FUNCTION_BLOCK Gerador (* CAT Gerador AGC150 - 15 blocos - 74 vars *)
  (* Standard: 61499-2 *)
  (* Version 7.0, 13/05/2026, Claude, 74 tags essenciais AGC150 *)
  PACKAGE Hidryco.HidrycoLib;
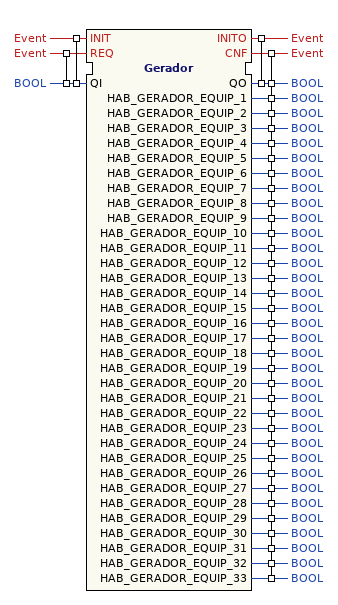
  EVENT_INPUT
    INIT WITH QI;
    REQ WITH QI;
  END_EVENT
  EVENT_OUTPUT
    INITO WITH QO;
    CNF WITH QO, HAB_GERADOR_EQUIP_4, HAB_GERADOR_EQUIP_5, HAB_GERADOR_EQUIP_6, HAB_GERADOR_EQUIP_7, HAB_GERADOR_EQUIP_8, HAB_GERADOR_EQUIP_9, HAB_GERADOR_EQUIP_10, HAB_GERADOR_EQUIP_11, HAB_GERADOR_EQUIP_12, HAB_GERADOR_EQUIP_13, HAB_GERADOR_EQUIP_14, HAB_GERADOR_EQUIP_15, HAB_GERADOR_EQUIP_16, HAB_GERADOR_EQUIP_17, HAB_GERADOR_EQUIP_18, HAB_GERADOR_EQUIP_19, HAB_GERADOR_EQUIP_20, HAB_GERADOR_EQUIP_21, HAB_GERADOR_EQUIP_22, HAB_GERADOR_EQUIP_23, HAB_GERADOR_EQUIP_24, HAB_GERADOR_EQUIP_25, HAB_GERADOR_EQUIP_26, HAB_GERADOR_EQUIP_27, HAB_GERADOR_EQUIP_28, HAB_GERADOR_EQUIP_29, HAB_GERADOR_EQUIP_30, HAB_GERADOR_EQUIP_31, HAB_GERADOR_EQUIP_32, HAB_GERADOR_EQUIP_33, HAB_GERADOR_EQUIP_1, HAB_GERADOR_EQUIP_2, HAB_GERADOR_EQUIP_3;
  END_EVENT
  VAR_INPUT
    QI : BOOL;
  END_VAR
  VAR_OUTPUT
    QO : BOOL;
    HAB_GERADOR_EQUIP_1 : BOOL; (* Habilitar equipamento 1 no gerador *)
    HAB_GERADOR_EQUIP_2 : BOOL; (* Habilitar equipamento 2 no gerador *)
    HAB_GERADOR_EQUIP_3 : BOOL; (* Habilitar equipamento 3 no gerador *)
    HAB_GERADOR_EQUIP_4 : BOOL; (* Habilitar equipamento 4 no gerador *)
    HAB_GERADOR_EQUIP_5 : BOOL; (* Habilitar equipamento 5 no gerador *)
    HAB_GERADOR_EQUIP_6 : BOOL; (* Habilitar equipamento 6 no gerador *)
    HAB_GERADOR_EQUIP_7 : BOOL; (* Habilitar equipamento 7 no gerador *)
    HAB_GERADOR_EQUIP_8 : BOOL; (* Habilitar equipamento 8 no gerador *)
    HAB_GERADOR_EQUIP_9 : BOOL; (* Habilitar equipamento 9 no gerador *)
    HAB_GERADOR_EQUIP_10 : BOOL; (* Habilitar equipamento 10 no gerador *)
    HAB_GERADOR_EQUIP_11 : BOOL; (* Habilitar equipamento 11 no gerador *)
    HAB_GERADOR_EQUIP_12 : BOOL; (* Habilitar equipamento 12 no gerador *)
    HAB_GERADOR_EQUIP_13 : BOOL; (* Habilitar equipamento 13 no gerador *)
    HAB_GERADOR_EQUIP_14 : BOOL; (* Habilitar equipamento 14 no gerador *)
    HAB_GERADOR_EQUIP_15 : BOOL; (* Habilitar equipamento 15 no gerador *)
    HAB_GERADOR_EQUIP_16 : BOOL; (* Habilitar equipamento 16 no gerador *)
    HAB_GERADOR_EQUIP_17 : BOOL; (* Habilitar equipamento 17 no gerador *)
    HAB_GERADOR_EQUIP_18 : BOOL; (* Habilitar equipamento 18 no gerador *)
    HAB_GERADOR_EQUIP_19 : BOOL; (* Habilitar equipamento 19 no gerador *)
    HAB_GERADOR_EQUIP_20 : BOOL; (* Habilitar equipamento 20 no gerador *)
    HAB_GERADOR_EQUIP_21 : BOOL; (* Habilitar equipamento 21 no gerador *)
    HAB_GERADOR_EQUIP_22 : BOOL; (* Habilitar equipamento 22 no gerador *)
    HAB_GERADOR_EQUIP_23 : BOOL; (* Habilitar equipamento 23 no gerador *)
    HAB_GERADOR_EQUIP_24 : BOOL; (* Habilitar equipamento 24 no gerador *)
    HAB_GERADOR_EQUIP_25 : BOOL; (* Habilitar equipamento 25 no gerador *)
    HAB_GERADOR_EQUIP_26 : BOOL; (* Habilitar equipamento 26 no gerador *)
    HAB_GERADOR_EQUIP_27 : BOOL; (* Habilitar equipamento 27 no gerador *)
    HAB_GERADOR_EQUIP_28 : BOOL; (* Habilitar equipamento 28 no gerador *)
    HAB_GERADOR_EQUIP_29 : BOOL; (* Habilitar equipamento 29 no gerador *)
    HAB_GERADOR_EQUIP_30 : BOOL; (* Habilitar equipamento 30 no gerador *)
    HAB_GERADOR_EQUIP_31 : BOOL; (* Habilitar equipamento 31 no gerador *)
    HAB_GERADOR_EQUIP_32 : BOOL; (* Habilitar equipamento 32 no gerador *)
    HAB_GERADOR_EQUIP_33 : BOOL; (* Habilitar equipamento 33 no gerador *)
  END_VAR
  FBS
    SL_DST_15INT_1 : SYMLINKMULTIVARDST_115C998103CD7017B(QI := TRUE, NAME1 := '$${PATH}Generator_voltage_L1L2', NAME2 := '$${PATH}Generator_voltage_L2L3', NAME3 := '$${PATH}Generator_voltage_L3L1', NAME4 := '$${PATH}Generator_voltage_L1N', NAME5 := '$${PATH}Generator_voltage_L2N', NAME6 := '$${PATH}Generator_voltage_L3N', NAME7 := '$${PATH}Generator_frequency_L1', NAME8 := '$${PATH}Generator_frequency_L2', NAME9 := '$${PATH}Generator_frequency_L3', NAME10 := '$${PATH}Generator_current_L1', NAME11 := '$${PATH}Generator_current_L2', NAME12 := '$${PATH}Generator_current_L3', NAME13 := '$${PATH}Generator_power_L1', NAME14 := '$${PATH}Generator_power_L2', NAME15 := '$${PATH}Generator_power_L3'); {SET_ATTRIBUTE(Configuration.GenericFBType.InterfaceParams, Runtime.System#I:=15;VALUE${I$}:INT,INT,INT,INT,INT,INT,INT,INT,INT,INT,INT,INT,INT,INT,INT)}
    SL_DST_15INT_2 : SYMLINKMULTIVARDST_115C998103CD7017B(QI := TRUE, NAME1 := '$${PATH}Generator_power', NAME2 := '$${PATH}Generator_reactive_power_L1', NAME3 := '$${PATH}Generator_reactive_power_L2', NAME4 := '$${PATH}Generator_reactive_power_L3', NAME5 := '$${PATH}Generator_reactive_power', NAME6 := '$${PATH}Generator_apparent_power_L1', NAME7 := '$${PATH}Generator_apparent_power_L2', NAME8 := '$${PATH}Generator_apparent_power_L3', NAME9 := '$${PATH}Generator_apparent_power', NAME10 := '$${PATH}Generator_PF', NAME11 := '$${PATH}Cosphi', NAME12 := '$${PATH}Cosphi_InductiveCapacitive_0Inductive_1C', NAME13 := '$${PATH}Generator_voltage_phase_angle_L1L2', NAME14 := '$${PATH}Generator_voltage_phase_angle_L2L3', NAME15 := '$${PATH}Generator_voltage_phase_angle_L3L1'); {SET_ATTRIBUTE(Configuration.GenericFBType.InterfaceParams, Runtime.System#I:=15;VALUE${I$}:INT,INT,INT,INT,INT,INT,INT,INT,INT,INT,INT,INT,INT,INT,INT)}
    SL_DST_15INT_3 : SYMLINKMULTIVARDST_115C998103CD7017B(QI := TRUE, NAME1 := '$${PATH}Rotacao_do_motor', NAME2 := '$${PATH}Temperatura_liq_arrefecimento', NAME3 := '$${PATH}Pressao_do_oleo_do_motor', NAME4 := '$${PATH}Temperatura_do_oleo_do_motor', NAME5 := '$${PATH}Temperatura_do_combustivel', NAME6 := '$${PATH}Temperatura_do_ar_de_admissao', NAME7 := '$${PATH}Nivel_do_liq_arrefecimento', NAME8 := '$${PATH}Consumo_de_combustivel', NAME9 := '$${PATH}Temp_coletor_de_admissao', NAME10 := '$${PATH}Carga_do_motor', NAME11 := '$${PATH}Temperatura_de_exaustao', NAME12 := '$${PATH}Horimetro_total_do_motor', NAME13 := '$${PATH}Tensao_da_bateria', NAME14 := '$${PATH}Nivel_de_oleo', NAME15 := '$${PATH}Temperatura_ambiente'); {SET_ATTRIBUTE(Configuration.GenericFBType.InterfaceParams, Runtime.System#I:=15;VALUE${I$}:INT,INT,INT,INT,INT,INT,INT,INT,INT,INT,INT,INT,INT,INT,INT)}
    SL_DST_4INT_4 : SYMLINKMULTIVARDST_15292F208F22048C1(QI := TRUE, NAME1 := '$${PATH}Combustivel_total_viagem', NAME2 := '$${PATH}Combustivel_total_acumulado', NAME3 := '$${PATH}Horas_de_funcionamento_absolutas', NAME4 := '$${PATH}Horas_de_funcionamento_relativas'); {SET_ATTRIBUTE(Configuration.GenericFBType.InterfaceParams, Runtime.System#I:=4;VALUE${I$}:INT,INT,INT,INT)}
    SL_DST_2INT_5 : SYMLINKMULTIVARDST_184BA62D721027C6E(QI := TRUE, NAME1 := '$${PATH}No_total_de_alarmes', NAME2 := '$${PATH}No_de_alarmes_nao_reconhecidos'); {SET_ATTRIBUTE(Configuration.GenericFBType.InterfaceParams, Runtime.System#I:=2;VALUE${I$}:INT,INT)}
    SL_DST_5BOOL_6 : SYMLINKMULTIVARDST_65D63179E2618F5E(QI := TRUE, NAME1 := '$${PATH}GB_position_ON', NAME2 := '$${PATH}MB_position_ON', NAME3 := '$${PATH}Running', NAME4 := '$${PATH}Generator_voltagefrequency_OK', NAME5 := '$${PATH}Mains_failure'); {SET_ATTRIBUTE(Configuration.GenericFBType.InterfaceParams, Runtime.System#I:=5;VALUE${I$}:BOOL,BOOL,BOOL,BOOL,BOOL)}
    SL_DST_5BOOL_7 : SYMLINKMULTIVARDST_65D63179E2618F5E(QI := TRUE, NAME1 := '$${PATH}Block_mode', NAME2 := '$${PATH}Manual_mode', NAME3 := '$${PATH}Semiauto_mode', NAME4 := '$${PATH}Auto_mode', NAME5 := '$${PATH}GB_position_OFF'); {SET_ATTRIBUTE(Configuration.GenericFBType.InterfaceParams, Runtime.System#I:=5;VALUE${I$}:BOOL,BOOL,BOOL,BOOL,BOOL)}
    SL_DST_1BOOL_8 : SYMLINKMULTIVARDST_1559B0FF8170C9BA0(QI := TRUE, NAME1 := '$${PATH}MB_position_OFF'); {SET_ATTRIBUTE(Configuration.GenericFBType.InterfaceParams, Runtime.System#I:=1;VALUE${I$}:BOOL)}
    SL_SRC_2BOOL_9 : SYMLINKMULTIVARSRC_277E97BEC1451D2C(QI := TRUE, NAME1 := '$${PATH}Remote_start', NAME2 := '$${PATH}Remote_stop'); {SET_ATTRIBUTE(Configuration.GenericFBType.InterfaceParams, Runtime.System#I:=2;VALUE${I$}:BOOL,BOOL)}
    SL_SRC_2BOOL_10 : SYMLINKMULTIVARSRC_277E97BEC1451D2C(QI := TRUE, NAME1 := '$${PATH}Remote_GB_ON', NAME2 := '$${PATH}Remote_GB_OFF'); {SET_ATTRIBUTE(Configuration.GenericFBType.InterfaceParams, Runtime.System#I:=2;VALUE${I$}:BOOL,BOOL)}
    SL_SRC_2BOOL_11 : SYMLINKMULTIVARSRC_277E97BEC1451D2C(QI := TRUE, NAME1 := '$${PATH}Start_sync', NAME2 := '$${PATH}Deload_stop'); {SET_ATTRIBUTE(Configuration.GenericFBType.InterfaceParams, Runtime.System#I:=2;VALUE${I$}:BOOL,BOOL)}
    SL_SRC_1BOOL_12 : SYMLINKMULTIVARSRC_1559B0FF8170C9BA0(QI := TRUE, NAME1 := '$${PATH}Test_mode_B15'); {SET_ATTRIBUTE(Configuration.GenericFBType.InterfaceParams, Runtime.System#I:=1;VALUE${I$}:BOOL)}
    SL_SRC_3INT_13 : SYMLINKMULTIVARSRC_154988C56DC16E7CE(QI := TRUE, NAME1 := '$${PATH}Setpoint_do_regulador_de_potencia_ativa', NAME2 := '$${PATH}Setpoint_cosPhi', NAME3 := '$${PATH}Setpoint_de_potencia_reativa'); {SET_ATTRIBUTE(Configuration.GenericFBType.InterfaceParams, Runtime.System#I:=3;VALUE${I$}:INT,INT,INT)}
    SL_SRC_1INT_14 : SYMLINKMULTIVARSRC_5A03F112CD5D470(QI := TRUE, NAME1 := '$${PATH}Setpoint_do_regulador_de_frequencia'); {SET_ATTRIBUTE(Configuration.GenericFBType.InterfaceParams, Runtime.System#I:=1;VALUE${I$}:INT)}
    SL_SRC_1INT_15 : SYMLINKMULTIVARSRC_5A03F112CD5D470(QI := TRUE, NAME1 := '$${PATH}Setpoint_do_regulador_de_tensao'); {SET_ATTRIBUTE(Configuration.GenericFBType.InterfaceParams, Runtime.System#I:=1;VALUE${I$}:INT)}
    IThis : Gerador_HMI(QI := TRUE);
    plcStart1 : plcStart;
    E_MERGE1 : E_MERGE;
    E_MERGE2 : E_MERGE;
    E_MERGE3 : E_MERGE;
    E_MERGE4 : E_MERGE;
    E_MERGE5 : E_MERGE;
    E_MERGE6 : E_MERGE;
    E_MERGE7 : E_MERGE;
    E_MERGE8 : E_MERGE;
    E_MERGE9 : E_MERGE;
    E_MERGE10 : E_MERGE;
    E_MERGE11 : E_MERGE;
    E_MERGE12 : E_MERGE;
    E_MERGE13 : E_MERGE;
    E_MERGE14 : E_MERGE;
    E_MERGE15 : E_MERGE;
    E_MERGE16 : E_MERGE;
    E_MERGE17 : E_MERGE;
    E_MERGE18 : E_MERGE;
    E_MERGE19 : E_MERGE;
    E_MERGE20 : E_MERGE;
    E_MERGE21 : E_MERGE;
    E_MERGE22 : E_MERGE;
    E_MERGE23 : E_MERGE;
    E_MERGE24 : E_MERGE;
    E_MERGE25 : E_MERGE;
    E_MERGE26 : E_MERGE;
    E_MERGE27 : E_MERGE;
    E_MERGE28 : E_MERGE;
    E_MERGE29 : E_MERGE;
    E_MERGE30 : E_MERGE;
    E_MERGE31 : E_MERGE;
    E_MERGE32 : E_MERGE;
  END_FBS
  EVENT_CONNECTIONS
    plcStart1.FIRST_INIT TO SL_DST_15INT_1.INIT;
    plcStart1.REDO_INIT TO SL_DST_15INT_1.INIT;
    SL_DST_15INT_1.INITO TO SL_DST_15INT_2.INIT;
    SL_DST_15INT_2.INITO TO SL_DST_15INT_3.INIT;
    SL_DST_15INT_3.INITO TO SL_DST_4INT_4.INIT;
    SL_DST_4INT_4.INITO TO SL_DST_2INT_5.INIT;
    SL_DST_2INT_5.INITO TO SL_DST_5BOOL_6.INIT;
    SL_DST_5BOOL_6.INITO TO SL_DST_5BOOL_7.INIT;
    SL_DST_5BOOL_7.INITO TO SL_DST_1BOOL_8.INIT;
    SL_DST_1BOOL_8.INITO TO SL_SRC_2BOOL_9.INIT;
    SL_SRC_2BOOL_9.INITO TO SL_SRC_2BOOL_10.INIT;
    SL_SRC_2BOOL_10.INITO TO SL_SRC_2BOOL_11.INIT;
    SL_SRC_2BOOL_11.INITO TO SL_SRC_1BOOL_12.INIT;
    SL_SRC_1BOOL_12.INITO TO SL_SRC_3INT_13.INIT;
    SL_SRC_3INT_13.INITO TO SL_SRC_1INT_14.INIT;
    SL_SRC_1INT_14.INITO TO SL_SRC_1INT_15.INIT;
    SL_SRC_1INT_15.INITO TO IThis.8F871B0D13D0118C;
    IThis.59C84A1FE88732D4 TO plcStart1.ACK_FIRST;
    SL_DST_15INT_1.CNF TO IThis.B45DE38A2141461E;
    SL_DST_15INT_2.CNF TO IThis.B45DE38A2141461E;
    SL_DST_15INT_3.CNF TO IThis.B45DE38A2141461E;
    SL_DST_4INT_4.CNF TO IThis.B45DE38A2141461E;
    SL_DST_2INT_5.CNF TO IThis.B45DE38A2141461E;
    SL_DST_5BOOL_6.CNF TO IThis.B45DE38A2141461E;
    SL_DST_5BOOL_7.CNF TO IThis.B45DE38A2141461E;
    SL_DST_1BOOL_8.CNF TO IThis.B45DE38A2141461E;
    IThis.6707C27F67701F0 TO SL_SRC_2BOOL_9.REQ;
    IThis.6707C27F67701F0 TO SL_SRC_2BOOL_10.REQ;
    IThis.6707C27F67701F0 TO SL_SRC_2BOOL_11.REQ;
    IThis.6707C27F67701F0 TO SL_SRC_1BOOL_12.REQ;
    IThis.6707C27F67701F0 TO SL_SRC_3INT_13.REQ;
    IThis.6707C27F67701F0 TO SL_SRC_1INT_14.REQ;
    IThis.6707C27F67701F0 TO SL_SRC_1INT_15.REQ;
    IThis.95A80690C09C71B3 TO SL_SRC_2BOOL_9.REQ;
    IThis.957FCC6414EC2F53 TO SL_SRC_2BOOL_9.REQ;
    IThis.4BB676D35CE52F17 TO SL_SRC_2BOOL_10.REQ;
    IThis.B47B8376792BFD25 TO SL_SRC_2BOOL_10.REQ;
    IThis.1E592EF8306DF830 TO SL_SRC_2BOOL_11.REQ;
    IThis.4E628C776CDEE1DA TO SL_SRC_2BOOL_11.REQ;
    IThis.4B9358773D12B730 TO E_MERGE1.EI1;
    IThis.78556F40A74B9612 TO E_MERGE1.EI2;
    E_MERGE1.EO TO E_MERGE2.EI1;
    IThis.B60DC44ACBE9CCB9 TO E_MERGE2.EI2;
    E_MERGE2.EO TO E_MERGE3.EI1;
    IThis.9AD02EE1BC3C744E TO E_MERGE3.EI2;
    E_MERGE3.EO TO E_MERGE4.EI1;
    IThis.D3249E894324CD69 TO E_MERGE4.EI2;
    E_MERGE5.EO TO E_MERGE6.EI1;
    E_MERGE6.EO TO E_MERGE7.EI1;
    E_MERGE7.EO TO E_MERGE8.EI1;
    E_MERGE4.EO TO E_MERGE5.EI1;
    IThis.641A9B22AD877AE1 TO E_MERGE5.EI2;
    IThis.DDB170EE3F1A0F27 TO E_MERGE6.EI2;
    IThis.FC8D521992645740 TO E_MERGE7.EI2;
    IThis.338BB6CD659261E7 TO E_MERGE8.EI2;
    E_MERGE9.EO TO E_MERGE10.EI1;
    E_MERGE10.EO TO E_MERGE11.EI1;
    E_MERGE11.EO TO E_MERGE12.EI1;
    E_MERGE13.EO TO E_MERGE14.EI1;
    E_MERGE14.EO TO E_MERGE15.EI1;
    E_MERGE15.EO TO E_MERGE16.EI1;
    E_MERGE12.EO TO E_MERGE13.EI1;
    E_MERGE8.EO TO E_MERGE9.EI1;
    IThis.2664114DEF28A59A TO E_MERGE9.EI2;
    IThis.A17221B212E515D0 TO E_MERGE10.EI2;
    IThis.67F8FA7A05619142 TO E_MERGE11.EI2;
    IThis.B073A3DCB15A968B TO E_MERGE12.EI2;
    IThis.98CBAE648FED4618 TO E_MERGE13.EI2;
    IThis.4E3FA93E68B940FC TO E_MERGE14.EI2;
    IThis.B6861634016BAF39 TO E_MERGE15.EI2;
    IThis.B354F41009F54AAE TO E_MERGE16.EI2;
    E_MERGE18.EO TO E_MERGE19.EI1;
    E_MERGE21.EO TO E_MERGE22.EI1;
    E_MERGE22.EO TO E_MERGE23.EI1;
    E_MERGE23.EO TO E_MERGE24.EI1;
    E_MERGE20.EO TO E_MERGE21.EI1;
    E_MERGE25.EO TO E_MERGE26.EI1;
    E_MERGE26.EO TO E_MERGE27.EI1;
    E_MERGE27.EO TO E_MERGE28.EI1;
    E_MERGE29.EO TO E_MERGE30.EI1;
    E_MERGE30.EO TO E_MERGE31.EI1;
    E_MERGE28.EO TO E_MERGE29.EI1;
    E_MERGE24.EO TO E_MERGE25.EI1;
    E_MERGE17.EO TO E_MERGE18.EI1;
    E_MERGE16.EO TO E_MERGE17.EI1;
    IThis.DC14AE43B9A5FB98 TO E_MERGE17.EI2;
    IThis.4EB1CCBB7A2E2865 TO E_MERGE18.EI2;
    IThis.02144F14BE588504 TO E_MERGE19.EI2;
    IThis.4DA3F4C465D1137C TO E_MERGE20.EI2;
    IThis.BA5363FBB7D30137 TO E_MERGE21.EI2;
    E_MERGE19.EO TO E_MERGE20.EI1;
    IThis.78DA1D0001F116A0 TO E_MERGE22.EI2;
    IThis.325C631DFC87D4F1 TO E_MERGE23.EI2;
    IThis.17F1D0A2267CBABA TO E_MERGE24.EI2;
    IThis.28629A0D2418E06B TO E_MERGE25.EI2;
    IThis.5E99AECC2045BAFC TO E_MERGE26.EI2;
    IThis.F15E09A4488D37F5 TO E_MERGE27.EI2;
    IThis.A650AAB0BDA0CE76 TO E_MERGE28.EI2;
    IThis.049966DDE656D0C4 TO E_MERGE29.EI2;
    IThis.5DC8F8B9CF00FC63 TO E_MERGE30.EI2;
    IThis.7DAE96B396D80193 TO E_MERGE31.EI2;
    IThis.B00AA3AD18EF7061 TO E_MERGE32.EI2;
    E_MERGE31.EO TO E_MERGE32.EI1;
    E_MERGE32.EO TO CNF;
  END_CONNECTIONS
  DATA_CONNECTIONS
    SL_DST_15INT_1.VALUE1 TO IThis.2DF05CC0E325A1EF;
    SL_DST_15INT_1.VALUE2 TO IThis.955D3B2CCB0C3B4A;
    SL_DST_15INT_1.VALUE3 TO IThis.C475E26CA9FEE82A;
    SL_DST_15INT_1.VALUE4 TO IThis.8C96B3395D200E1C;
    SL_DST_15INT_1.VALUE5 TO IThis.F357E24BA3D817DB;
    SL_DST_15INT_1.VALUE6 TO IThis.5022D3AA4F4D90E9;
    SL_DST_15INT_1.VALUE7 TO IThis.AB616A18FAEDD063;
    SL_DST_15INT_1.VALUE8 TO IThis.90079364ED2A2AEE;
    SL_DST_15INT_1.VALUE9 TO IThis.1A02B46DCB3CD9A8;
    SL_DST_15INT_1.VALUE10 TO IThis.E5CD34123669C031;
    SL_DST_15INT_1.VALUE11 TO IThis.86247BDAA3CA16FE;
    SL_DST_15INT_1.VALUE12 TO IThis.2C1D109D343C43A8;
    SL_DST_15INT_1.VALUE13 TO IThis.48ECE1C0CDB3B0D3;
    SL_DST_15INT_1.VALUE14 TO IThis.C6EB5487BD84797B;
    SL_DST_15INT_1.VALUE15 TO IThis.807575BFFC1B7A6B;
    SL_DST_15INT_2.VALUE1 TO IThis.5DE20FA101C23950;
    SL_DST_15INT_2.VALUE2 TO IThis.E44A7D858964B0B3;
    SL_DST_15INT_2.VALUE3 TO IThis.F28A918593FB105D;
    SL_DST_15INT_2.VALUE4 TO IThis.3CED272C8ACF0A7C;
    SL_DST_15INT_2.VALUE5 TO IThis.A438FE13D9E8A7F5;
    SL_DST_15INT_2.VALUE6 TO IThis.22833FD3EDA77F7D;
    SL_DST_15INT_2.VALUE7 TO IThis.49E2125CAA7ECCA1;
    SL_DST_15INT_2.VALUE8 TO IThis.8CCFFAF45EC352B2;
    SL_DST_15INT_2.VALUE9 TO IThis.7EF881336FCA17EF;
    SL_DST_15INT_2.VALUE10 TO IThis.7EE19F4B6530CD29;
    SL_DST_15INT_2.VALUE11 TO IThis.8D98BD9709ACA518;
    SL_DST_15INT_2.VALUE12 TO IThis.DBA74DB3B3605E26;
    SL_DST_15INT_2.VALUE13 TO IThis.F53E7A129A9A0A2C;
    SL_DST_15INT_2.VALUE14 TO IThis.183E9D0116DFBB48;
    SL_DST_15INT_2.VALUE15 TO IThis.6BAC6C6020DE83F6;
    SL_DST_15INT_3.VALUE1 TO IThis.DFEBF0ED41045FE9;
    SL_DST_15INT_3.VALUE2 TO IThis.F393DADE5A3CB254;
    SL_DST_15INT_3.VALUE3 TO IThis.750F0479BAF5EF07;
    SL_DST_15INT_3.VALUE4 TO IThis.AA1A8607FA552EA4;
    SL_DST_15INT_3.VALUE5 TO IThis.C58EBBC0A647B0AB;
    SL_DST_15INT_3.VALUE6 TO IThis.7E9AD6DEEE5B52E7;
    SL_DST_15INT_3.VALUE7 TO IThis.7410C12C9A19F1F;
    SL_DST_15INT_3.VALUE8 TO IThis.8F185C4AB29E91B4;
    SL_DST_15INT_3.VALUE9 TO IThis.1119A8BA2959E489;
    SL_DST_15INT_3.VALUE10 TO IThis.ABDAA0D2A934F3EC;
    SL_DST_15INT_3.VALUE11 TO IThis.CC4858EEA998D695;
    SL_DST_15INT_3.VALUE12 TO IThis.D75494F989FCA7ED;
    SL_DST_15INT_3.VALUE13 TO IThis.3D3695A828CE84AB;
    SL_DST_15INT_3.VALUE14 TO IThis.5DFE63F451819395;
    SL_DST_15INT_3.VALUE15 TO IThis.8CFF3BEB9D2FAAD;
    SL_DST_4INT_4.VALUE1 TO IThis.9405FC1C00A32AEC;
    SL_DST_4INT_4.VALUE2 TO IThis.2B5FBEB04594604E;
    SL_DST_4INT_4.VALUE3 TO IThis.120D763B5AD8C720;
    SL_DST_4INT_4.VALUE4 TO IThis.1073690F8B08618C;
    SL_DST_2INT_5.VALUE1 TO IThis.C9AE3A5F75F27009;
    SL_DST_2INT_5.VALUE2 TO IThis.F31C547F2345F058;
    SL_DST_5BOOL_6.VALUE1 TO IThis.440C5F1A46820EA9;
    SL_DST_5BOOL_6.VALUE3 TO IThis.B44A610B1AC7DDCB;
    SL_DST_5BOOL_6.VALUE4 TO IThis.89E752459C0DB9D;
    SL_DST_5BOOL_6.VALUE5 TO IThis.A1ED45F6761341C9;
    SL_DST_5BOOL_7.VALUE1 TO IThis.EBF6FFCF6E686E61;
    SL_DST_5BOOL_7.VALUE2 TO IThis.F01721D461BE15D1;
    SL_DST_5BOOL_7.VALUE3 TO IThis.279E7F947F480A6B;
    SL_DST_5BOOL_7.VALUE4 TO IThis.EAF6D802ADD9C5EC;
    SL_DST_5BOOL_7.VALUE5 TO IThis.C3459D671815F793;
    IThis.D267C42A1DA85017 TO SL_SRC_2BOOL_9.VALUE1;
    IThis.B6AF108F10E5C7B9 TO SL_SRC_2BOOL_9.VALUE2;
    IThis.AD9FA969B8F910CF TO SL_SRC_2BOOL_10.VALUE1;
    IThis.50C247679F4E3A6F TO SL_SRC_2BOOL_10.VALUE2;
    IThis.CFC5C61590EC7393 TO SL_SRC_2BOOL_11.VALUE1;
    IThis.63A01CA214EE4F9E TO SL_SRC_2BOOL_11.VALUE2;
    IThis.199F97C8DC275581 TO SL_SRC_3INT_13.VALUE1;
    IThis.94D1A6DB5D930DEE TO SL_SRC_3INT_13.VALUE2;
    IThis.F01298F98FD57660 TO SL_SRC_3INT_13.VALUE3;
    IThis.984CCD272C02FB1E TO SL_SRC_1INT_14.VALUE1;
    IThis.8274CD43C7386532 TO SL_SRC_1INT_15.VALUE1;
    IThis.44EF2CBDCBF3D63B TO HAB_GERADOR_EQUIP_1;
    IThis.849F0F311619FDBB TO HAB_GERADOR_EQUIP_2;
    IThis.108E878CDC776750 TO HAB_GERADOR_EQUIP_3;
    IThis.C90E3681A8307381 TO HAB_GERADOR_EQUIP_33;
    IThis.C929428314AF7B70 TO HAB_GERADOR_EQUIP_32;
    IThis.3C23406B0BA5381A TO HAB_GERADOR_EQUIP_31;
    IThis.DF5F9409B2EEC4D9 TO HAB_GERADOR_EQUIP_30;
    IThis.1552D3BF196D22A4 TO HAB_GERADOR_EQUIP_29;
    IThis.A70B738B6E050E17 TO HAB_GERADOR_EQUIP_28;
    IThis.169E06199FCE9259 TO HAB_GERADOR_EQUIP_27;
    IThis.405056098285C3A4 TO HAB_GERADOR_EQUIP_26;
    IThis.72968085D7C95002 TO HAB_GERADOR_EQUIP_25;
    IThis.C12D0B7C80F94596 TO HAB_GERADOR_EQUIP_24;
    IThis.F0D74C2F7205767B TO HAB_GERADOR_EQUIP_23;
    IThis.D9D6D2D7835B7E40 TO HAB_GERADOR_EQUIP_22;
    IThis.D248E3F6C6054B9A TO HAB_GERADOR_EQUIP_21;
    IThis.F30FB4F377AC3E75 TO HAB_GERADOR_EQUIP_20;
    IThis.87E506DF7C28048B TO HAB_GERADOR_EQUIP_19;
    IThis.658BA795C10DFD8C TO HAB_GERADOR_EQUIP_18;
    IThis.2D3AB65C79025B8E TO HAB_GERADOR_EQUIP_17;
    IThis.1C7A46DADC6E29DF TO HAB_GERADOR_EQUIP_16;
    IThis.DCAA3C9A253B06CD TO HAB_GERADOR_EQUIP_15;
    IThis.7DA84572FCC76F28 TO HAB_GERADOR_EQUIP_14;
    IThis.09981BB9828BA6DE TO HAB_GERADOR_EQUIP_13;
    IThis.6A26AFC1C110D8DE TO HAB_GERADOR_EQUIP_12;
    IThis.422878E19F89E778 TO HAB_GERADOR_EQUIP_11;
    IThis.1B28BDD327EBC80C TO HAB_GERADOR_EQUIP_10;
    IThis.BC96A9D59C810BF7 TO HAB_GERADOR_EQUIP_9;
    IThis.3188B3A04DFEB842 TO HAB_GERADOR_EQUIP_8;
    IThis.526E1B4971AD2247 TO HAB_GERADOR_EQUIP_7;
    IThis.3C1A45957510E720 TO HAB_GERADOR_EQUIP_6;
    IThis.046F77AFACED4554 TO HAB_GERADOR_EQUIP_5;
    IThis.CC738ED511BCD0B9 TO HAB_GERADOR_EQUIP_4;
  END_CONNECTIONS
END_FUNCTION_BLOCK
